// TIA Portal V16 export
// export: Created 2022-03-28T07:44:06.5972207Z, ExportSetting WithDefaults, DisplayName Totally Integrated Automation Portal, DisplayVersion V16 Update 5, DisplayName TIA Portal Version Control Interface, DisplayVersion V16 Update 2, DisplayName TIA Portal Openness, DisplayVersion V16 Update 5, DisplayName STEP 7 Professional, DisplayVersion V16 Update 5, DisplayName STEP 7 Safety, DisplayVersion V16, DisplayName WinCC Professional, DisplayVersion V16 Update 5
FUNCTION_BLOCK "fb_01_Cycle"   // FB1, LAD
{ S7_Optimized_Access := 'TRUE' }
VERSION : 0.1
// stored: AutoNumber false, IsIECCheckEnabled false, IsRetainMemResEnabled false, MemoryReserve 100, SetENOAutomatically false, UDAEnableTagReadback false
   VAR
      TON_Delay : Array[1..10] of TON_TIME;
      TP_Reset { S7_SetPoint := 'True'} : TP_TIME;
   END_VAR
   VAR_TEMP
      bBypassRobot : Bool;
      bRobotReset : Bool;
      bIsInverted : Bool;
   END_VAR
   VAR_TEMP   // added for the SCL form of the ladder/FBD networks
      _w1 : Bool;
      _w2 : Bool;
   END_VAR
BEGIN

REGION Network 1: Reseteo Ciclos por Emergencias
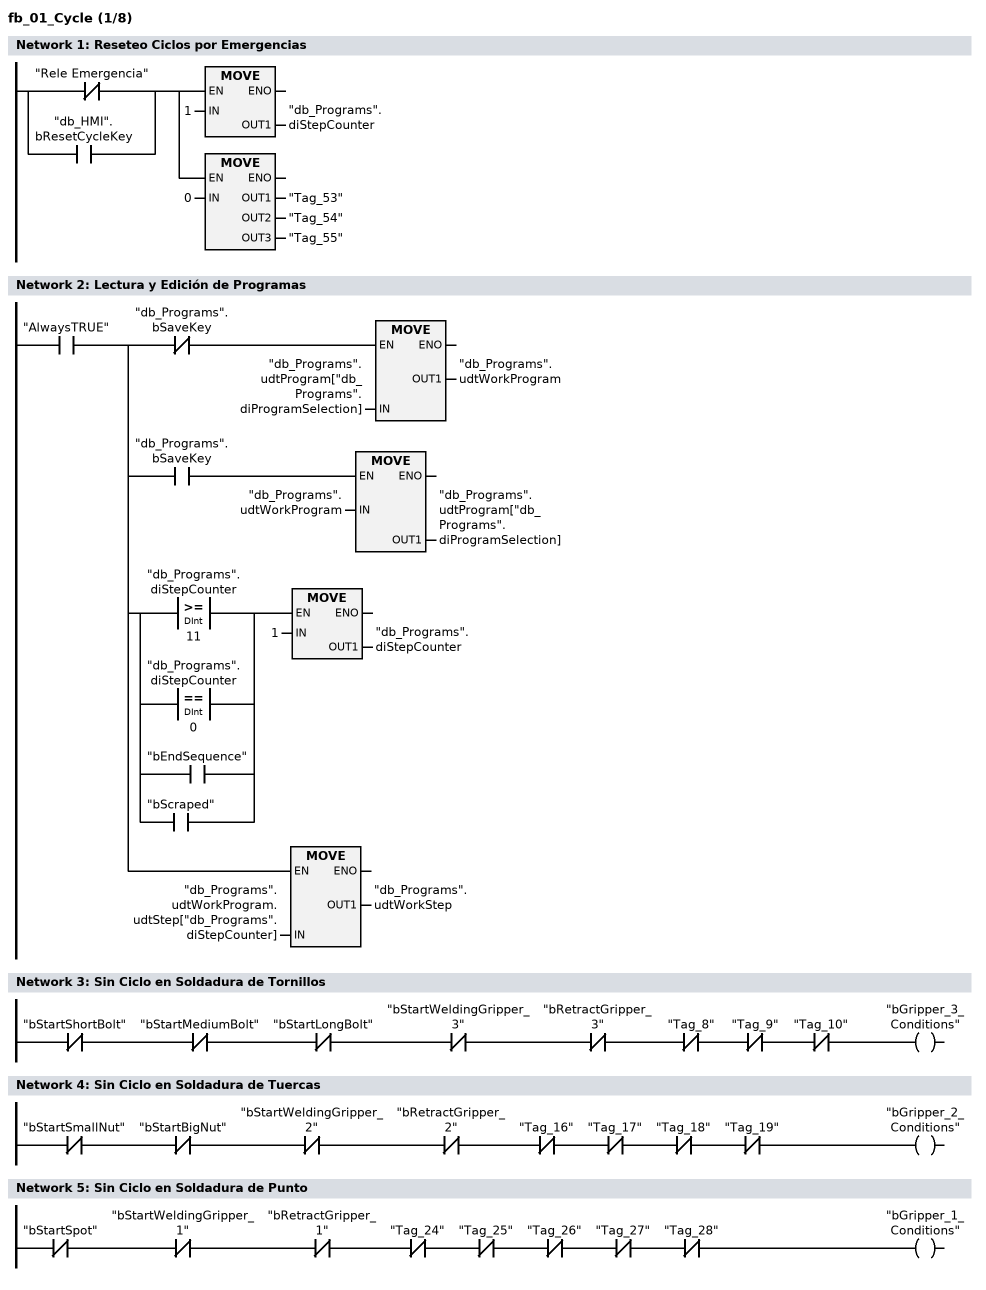
   RUNG wire#powerrail
      I_Contact( "Rele Emergencia" )
      wire#w1
      Move(in := 1, out1 => "db_Programs".diStepCounter)
   END_RUNG
   RUNG wire#powerrail
      Contact( "db_HMI".bResetCycleKey )
   END_RUNG wire#w1
   RUNG wire#w1
      Move(in := 0, out1 => "Tag_53", out2 => "Tag_54", out3 => "Tag_55")
   END_RUNG
   // the same network as SCL:
   IF NOT "Rele Emergencia" OR "db_HMI".bResetCycleKey THEN
       "db_Programs".diStepCounter := 1;
       "Tag_53" := 0;
       "Tag_54" := 0;
       "Tag_55" := 0;
   END_IF;
END_REGION

REGION Network 2: Lectura y Edición de Programas
   RUNG wire#powerrail
      Contact( "AlwaysTRUE" )
      wire#w1
      I_Contact( "db_Programs".bSaveKey )
      Move(in := "db_Programs".udtProgram["db_Programs".diProgramSelection], out1 => "db_Programs".udtWorkProgram)
   END_RUNG
   RUNG wire#w1
      Contact( "db_Programs".bSaveKey )
      Move(in := "db_Programs".udtWorkProgram, out1 => "db_Programs".udtProgram["db_Programs".diProgramSelection])
   END_RUNG
   RUNG wire#w1
      { S7_Templates := "SrcType := DInt" } GE_Contact(in1 := "db_Programs".diStepCounter, in2 := 11)
      wire#w2
      Move(in := 1, out1 => "db_Programs".diStepCounter)
   END_RUNG
   RUNG wire#w1
      { S7_Templates := "SrcType := DInt" } EQ_Contact(in1 := "db_Programs".diStepCounter, in2 := 0)
   END_RUNG wire#w2
   RUNG wire#w1
      Contact( "bEndSequence" )
   END_RUNG wire#w2
   RUNG wire#w1
      Contact( "bScraped" )
   END_RUNG wire#w2
   RUNG wire#w1
      Move(in := "db_Programs".udtWorkProgram.udtStep["db_Programs".diStepCounter], out1 => "db_Programs".udtWorkStep)
   END_RUNG
   // the same network as SCL:
   IF "AlwaysTRUE" AND NOT "db_Programs".bSaveKey THEN
       "db_Programs".udtWorkProgram := "db_Programs".udtProgram["db_Programs".diProgramSelection];
   END_IF;
   IF "AlwaysTRUE" AND "db_Programs".bSaveKey THEN
       "db_Programs".udtProgram["db_Programs".diProgramSelection] := "db_Programs".udtWorkProgram;
   END_IF;
   IF "AlwaysTRUE" AND (("db_Programs".diStepCounter >= 11) OR ("db_Programs".diStepCounter = 0) OR "bEndSequence" OR "bScraped") THEN
       "db_Programs".diStepCounter := 1;
   END_IF;
   IF "AlwaysTRUE" THEN
       "db_Programs".udtWorkStep := "db_Programs".udtWorkProgram.udtStep["db_Programs".diStepCounter];
   END_IF;
END_REGION

REGION Network 3: Sin Ciclo en Soldadura de Tornillos
   RUNG wire#powerrail
      I_Contact( "bStartShortBolt" )
      I_Contact( "bStartMediumBolt" )
      I_Contact( "bStartLongBolt" )
      I_Contact( "bStartWeldingGripper_3" )
      I_Contact( "bRetractGripper_3" )
      I_Contact( "Tag_8" )
      I_Contact( "Tag_9" )
      I_Contact( "Tag_10" )
      Coil( "bGripper_3_Conditions" )
   END_RUNG
   // the same network as SCL:
   "bGripper_3_Conditions" := NOT "bStartShortBolt" AND NOT "bStartMediumBolt" AND NOT "bStartLongBolt" AND NOT "bStartWeldingGripper_3" AND NOT "bRetractGripper_3" AND NOT "Tag_8" AND NOT "Tag_9" AND NOT "Tag_10";
END_REGION

REGION Network 4: Sin Ciclo en Soldadura de Tuercas
   RUNG wire#powerrail
      I_Contact( "bStartSmallNut" )
      I_Contact( "bStartBigNut" )
      I_Contact( "bStartWeldingGripper_2" )
      I_Contact( "bRetractGripper_2" )
      I_Contact( "Tag_16" )
      I_Contact( "Tag_17" )
      I_Contact( "Tag_18" )
      I_Contact( "Tag_19" )
      Coil( "bGripper_2_Conditions" )
   END_RUNG
   // the same network as SCL:
   "bGripper_2_Conditions" := NOT "bStartSmallNut" AND NOT "bStartBigNut" AND NOT "bStartWeldingGripper_2" AND NOT "bRetractGripper_2" AND NOT "Tag_16" AND NOT "Tag_17" AND NOT "Tag_18" AND NOT "Tag_19";
END_REGION

REGION Network 5: Sin Ciclo en Soldadura de Punto
   RUNG wire#powerrail
      I_Contact( "bStartSpot" )
      I_Contact( "bStartWeldingGripper_1" )
      I_Contact( "bRetractGripper_1" )
      I_Contact( "Tag_24" )
      I_Contact( "Tag_25" )
      I_Contact( "Tag_26" )
      I_Contact( "Tag_27" )
      I_Contact( "Tag_28" )
      Coil( "bGripper_1_Conditions" )
   END_RUNG
   // the same network as SCL:
   "bGripper_1_Conditions" := NOT "bStartSpot" AND NOT "bStartWeldingGripper_1" AND NOT "bRetractGripper_1" AND NOT "Tag_24" AND NOT "Tag_25" AND NOT "Tag_26" AND NOT "Tag_27" AND NOT "Tag_28";
END_REGION

REGION Network 6: Condiciones Ciclo Auxiliares
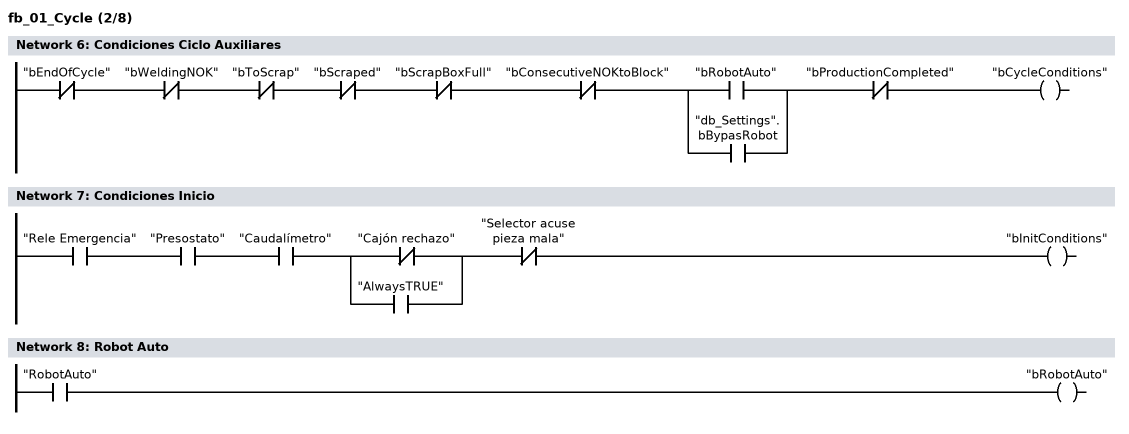
   RUNG wire#powerrail
      I_Contact( "bEndOfCycle" )
      I_Contact( "bWeldingNOK" )
      I_Contact( "bToScrap" )
      I_Contact( "bScraped" )
      I_Contact( "bScrapBoxFull" )
      I_Contact( "bConsecutiveNOKtoBlock" )
      wire#w1
      Contact( "bRobotAuto" )
      wire#w2
      I_Contact( "bProductionCompleted" )
      Coil( "bCycleConditions" )
   END_RUNG
   RUNG wire#w1
      Contact( "db_Settings".bBypasRobot )
   END_RUNG wire#w2
   // the same network as SCL:
   "bCycleConditions" := NOT "bEndOfCycle" AND NOT "bWeldingNOK" AND NOT "bToScrap" AND NOT "bScraped" AND NOT "bScrapBoxFull" AND NOT "bConsecutiveNOKtoBlock" AND ("bRobotAuto" OR "db_Settings".bBypasRobot) AND NOT "bProductionCompleted";
END_REGION

REGION Network 7: Condiciones Inicio
   RUNG wire#powerrail
      Contact( "Rele Emergencia" )
      Contact( "Presostato" )
      Contact( "Caudalímetro" )
      wire#w1
      I_Contact( "Cajón rechazo" )
      wire#w2
      I_Contact( "Selector acuse pieza mala" )
      Coil( "bInitConditions" )
   END_RUNG
   RUNG wire#w1
      Contact( "AlwaysTRUE" )
   END_RUNG wire#w2
   // the same network as SCL:
   "bInitConditions" := "Rele Emergencia" AND "Presostato" AND "Caudalímetro" AND (NOT "Cajón rechazo" OR "AlwaysTRUE") AND NOT "Selector acuse pieza mala";
END_REGION

REGION Network 8: Robot Auto
   RUNG wire#powerrail
      Contact( "RobotAuto" )
      Coil( "bRobotAuto" )
   END_RUNG
   // the same network as SCL:
   "bRobotAuto" := "RobotAuto";
END_REGION

REGION Network 9: Selección Acción
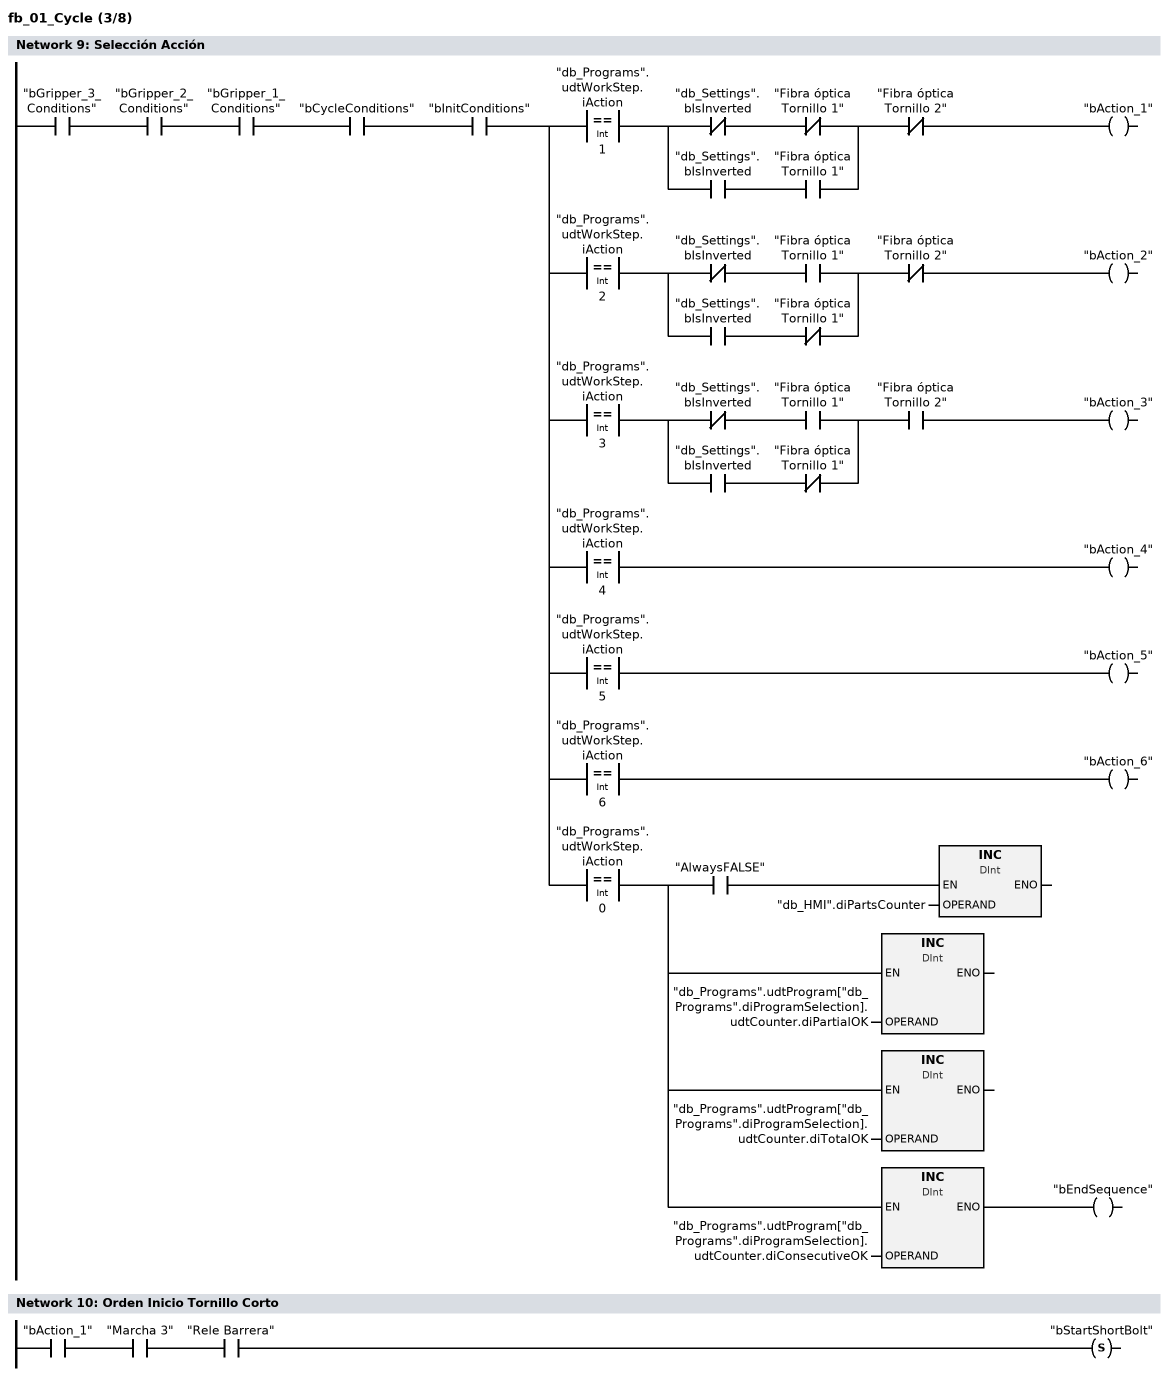
   RUNG wire#powerrail
      Contact( "bGripper_3_Conditions" )
      Contact( "bGripper_2_Conditions" )
      Contact( "bGripper_1_Conditions" )
      Contact( "bCycleConditions" )
      Contact( "bInitConditions" )
      wire#w1
      { S7_Templates := "SrcType := Int" } EQ_Contact(in1 := "db_Programs".udtWorkStep.iAction, in2 := 1)
      wire#w2
      I_Contact( "db_Settings".bIsInverted )
      I_Contact( "Fibra óptica Tornillo 1" )
      wire#w3
      I_Contact( "Fibra óptica Tornillo 2" )
      Coil( "bAction_1" )
   END_RUNG
   RUNG wire#w2
      Contact( "db_Settings".bIsInverted )
      Contact( "Fibra óptica Tornillo 1" )
   END_RUNG wire#w3
   RUNG wire#w1
      { S7_Templates := "SrcType := Int" } EQ_Contact(in1 := "db_Programs".udtWorkStep.iAction, in2 := 2)
      wire#w4
      I_Contact( "db_Settings".bIsInverted )
      Contact( "Fibra óptica Tornillo 1" )
      wire#w5
      I_Contact( "Fibra óptica Tornillo 2" )
      Coil( "bAction_2" )
   END_RUNG
   RUNG wire#w4
      Contact( "db_Settings".bIsInverted )
      I_Contact( "Fibra óptica Tornillo 1" )
   END_RUNG wire#w5
   RUNG wire#w1
      { S7_Templates := "SrcType := Int" } EQ_Contact(in1 := "db_Programs".udtWorkStep.iAction, in2 := 3)
      wire#w6
      I_Contact( "db_Settings".bIsInverted )
      Contact( "Fibra óptica Tornillo 1" )
      wire#w7
      Contact( "Fibra óptica Tornillo 2" )
      Coil( "bAction_3" )
   END_RUNG
   RUNG wire#w6
      Contact( "db_Settings".bIsInverted )
      I_Contact( "Fibra óptica Tornillo 1" )
   END_RUNG wire#w7
   RUNG wire#w1
      { S7_Templates := "SrcType := Int" } EQ_Contact(in1 := "db_Programs".udtWorkStep.iAction, in2 := 4)
      Coil( "bAction_4" )
   END_RUNG
   RUNG wire#w1
      { S7_Templates := "SrcType := Int" } EQ_Contact(in1 := "db_Programs".udtWorkStep.iAction, in2 := 5)
      Coil( "bAction_5" )
   END_RUNG
   RUNG wire#w1
      { S7_Templates := "SrcType := Int" } EQ_Contact(in1 := "db_Programs".udtWorkStep.iAction, in2 := 6)
      Coil( "bAction_6" )
   END_RUNG
   RUNG wire#w1
      { S7_Templates := "SrcType := Int" } EQ_Contact(in1 := "db_Programs".udtWorkStep.iAction, in2 := 0)
      wire#w8
      Contact( "AlwaysFALSE" )
      { S7_Templates := "DestType := DInt" } Inc( "db_HMI".diPartsCounter )
   END_RUNG
   RUNG wire#w8
      { S7_Templates := "DestType := DInt" } Inc( "db_Programs".udtProgram["db_Programs".diProgramSelection].udtCounter.diPartialOK )
   END_RUNG
   RUNG wire#w8
      { S7_Templates := "DestType := DInt" } Inc( "db_Programs".udtProgram["db_Programs".diProgramSelection].udtCounter.diTotalOK )
   END_RUNG
   RUNG wire#w8
      { S7_Templates := "DestType := DInt" } Inc( "db_Programs".udtProgram["db_Programs".diProgramSelection].udtCounter.diConsecutiveOK )
      Coil( "bEndSequence" )
   END_RUNG
   // the same network as SCL:
   #_w1 := "bGripper_3_Conditions" AND "bGripper_2_Conditions" AND "bGripper_1_Conditions" AND "bCycleConditions" AND "bInitConditions";
   "bAction_1" := #_w1 AND ("db_Programs".udtWorkStep.iAction = 1) AND ((NOT "db_Settings".bIsInverted AND NOT "Fibra óptica Tornillo 1") OR ("db_Settings".bIsInverted AND "Fibra óptica Tornillo 1")) AND NOT "Fibra óptica Tornillo 2";
   "bAction_2" := #_w1 AND ("db_Programs".udtWorkStep.iAction = 2) AND ((NOT "db_Settings".bIsInverted AND "Fibra óptica Tornillo 1") OR ("db_Settings".bIsInverted AND NOT "Fibra óptica Tornillo 1")) AND NOT "Fibra óptica Tornillo 2";
   "bAction_3" := #_w1 AND ("db_Programs".udtWorkStep.iAction = 3) AND ((NOT "db_Settings".bIsInverted AND "Fibra óptica Tornillo 1") OR ("db_Settings".bIsInverted AND NOT "Fibra óptica Tornillo 1")) AND "Fibra óptica Tornillo 2";
   "bAction_4" := #_w1 AND ("db_Programs".udtWorkStep.iAction = 4);
   "bAction_5" := #_w1 AND ("db_Programs".udtWorkStep.iAction = 5);
   "bAction_6" := #_w1 AND ("db_Programs".udtWorkStep.iAction = 6);
   #_w2 := #_w1 AND ("db_Programs".udtWorkStep.iAction = 0);
   IF #_w2 AND "AlwaysFALSE" THEN "db_HMI".diPartsCounter := "db_HMI".diPartsCounter + 1; END_IF;
   IF #_w2 THEN
       "db_Programs".udtProgram["db_Programs".diProgramSelection].udtCounter.diPartialOK := "db_Programs".udtProgram["db_Programs".diProgramSelection].udtCounter.diPartialOK + 1;
       "db_Programs".udtProgram["db_Programs".diProgramSelection].udtCounter.diTotalOK := "db_Programs".udtProgram["db_Programs".diProgramSelection].udtCounter.diTotalOK + 1;
       "db_Programs".udtProgram["db_Programs".diProgramSelection].udtCounter.diConsecutiveOK := "db_Programs".udtProgram["db_Programs".diProgramSelection].udtCounter.diConsecutiveOK + 1;
   END_IF;
   "bEndSequence" := #_w2;
END_REGION

REGION Network 10: Orden Inicio Tornillo Corto
   RUNG wire#powerrail
      Contact( "bAction_1" )
      Contact( "Marcha 3" )
      Contact( "Rele Barrera" )
      S_Coil( "bStartShortBolt" )
   END_RUNG
   // the same network as SCL:
   IF "bAction_1" AND "Marcha 3" AND "Rele Barrera" THEN "bStartShortBolt" := TRUE; END_IF;
END_REGION

REGION Network 11: Orden Inicio Tornillo Mediano
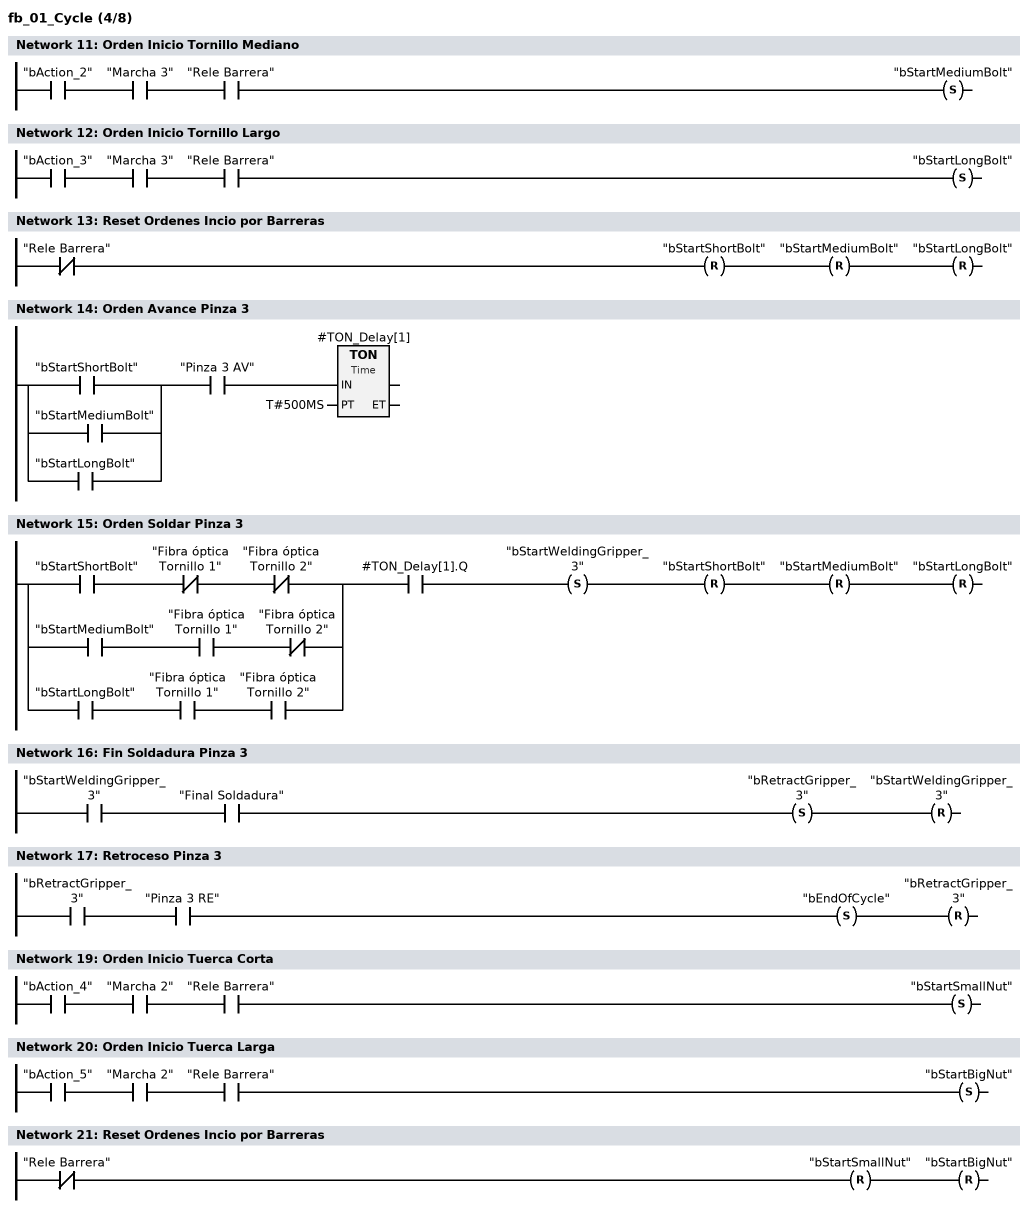
   RUNG wire#powerrail
      Contact( "bAction_2" )
      Contact( "Marcha 3" )
      Contact( "Rele Barrera" )
      S_Coil( "bStartMediumBolt" )
   END_RUNG
   // the same network as SCL:
   IF "bAction_2" AND "Marcha 3" AND "Rele Barrera" THEN "bStartMediumBolt" := TRUE; END_IF;
END_REGION

REGION Network 12: Orden Inicio Tornillo Largo
   RUNG wire#powerrail
      Contact( "bAction_3" )
      Contact( "Marcha 3" )
      Contact( "Rele Barrera" )
      S_Coil( "bStartLongBolt" )
   END_RUNG
   // the same network as SCL:
   IF "bAction_3" AND "Marcha 3" AND "Rele Barrera" THEN "bStartLongBolt" := TRUE; END_IF;
END_REGION

REGION Network 13: Reset Ordenes Incio por Barreras
   RUNG wire#powerrail
      I_Contact( "Rele Barrera" )
      R_Coil( "bStartShortBolt" )
      R_Coil( "bStartMediumBolt" )
      R_Coil( "bStartLongBolt" )
   END_RUNG
   // the same network as SCL:
   IF NOT "Rele Barrera" THEN
       "bStartShortBolt" := FALSE;
       "bStartMediumBolt" := FALSE;
       "bStartLongBolt" := FALSE;
   END_IF;
END_REGION

REGION Network 14: Orden Avance Pinza 3
   RUNG wire#powerrail
      Contact( "bStartShortBolt" )
      wire#w1
      Contact( "Pinza 3 AV" )
      { S7_Templates := "time_type := Time" } #TON_Delay[1].TON(pt := T#500MS, et =>)
   END_RUNG
   RUNG wire#powerrail
      Contact( "bStartMediumBolt" )
   END_RUNG wire#w1
   RUNG wire#powerrail
      Contact( "bStartLongBolt" )
   END_RUNG wire#w1
   // the same network as SCL:
   #TON_Delay[1].TON(IN := ("bStartShortBolt" OR "bStartMediumBolt" OR "bStartLongBolt") AND "Pinza 3 AV",
                     PT := T#500MS);
END_REGION

REGION Network 15: Orden Soldar Pinza 3
   RUNG wire#powerrail
      Contact( "bStartShortBolt" )
      I_Contact( "Fibra óptica Tornillo 1" )
      I_Contact( "Fibra óptica Tornillo 2" )
      wire#w1
      Contact( #TON_Delay[1].Q )
      S_Coil( "bStartWeldingGripper_3" )
      R_Coil( "bStartShortBolt" )
      R_Coil( "bStartMediumBolt" )
      R_Coil( "bStartLongBolt" )
   END_RUNG
   RUNG wire#powerrail
      Contact( "bStartMediumBolt" )
      Contact( "Fibra óptica Tornillo 1" )
      I_Contact( "Fibra óptica Tornillo 2" )
   END_RUNG wire#w1
   RUNG wire#powerrail
      Contact( "bStartLongBolt" )
      Contact( "Fibra óptica Tornillo 1" )
      Contact( "Fibra óptica Tornillo 2" )
   END_RUNG wire#w1
   // the same network as SCL:
   IF (("bStartShortBolt" AND NOT "Fibra óptica Tornillo 1" AND NOT "Fibra óptica Tornillo 2") OR ("bStartMediumBolt" AND "Fibra óptica Tornillo 1" AND NOT "Fibra óptica Tornillo 2") OR ("bStartLongBolt" AND "Fibra óptica Tornillo 1" AND "Fibra óptica Tornillo 2")) AND #TON_Delay[1].Q THEN
       "bStartWeldingGripper_3" := TRUE;
   END_IF;
   #_w1 := (("bStartShortBolt" AND NOT "Fibra óptica Tornillo 1" AND NOT "Fibra óptica Tornillo 2") OR ("bStartMediumBolt" AND "Fibra óptica Tornillo 1" AND NOT "Fibra óptica Tornillo 2") OR ("bStartLongBolt" AND "Fibra óptica Tornillo 1" AND "Fibra óptica Tornillo 2")) AND #TON_Delay[1].Q;
   IF #_w1 THEN
       "bStartShortBolt" := FALSE;
       "bStartMediumBolt" := FALSE;
       "bStartLongBolt" := FALSE;
   END_IF;
END_REGION

REGION Network 16: Fin Soldadura Pinza 3
   RUNG wire#powerrail
      Contact( "bStartWeldingGripper_3" )
      Contact( "Final Soldadura" )
      S_Coil( "bRetractGripper_3" )
      R_Coil( "bStartWeldingGripper_3" )
   END_RUNG
   // the same network as SCL:
   IF "bStartWeldingGripper_3" AND "Final Soldadura" THEN
       "bRetractGripper_3" := TRUE;
       "bStartWeldingGripper_3" := FALSE;
   END_IF;
END_REGION

REGION Network 17: Retroceso Pinza 3
   RUNG wire#powerrail
      Contact( "bRetractGripper_3" )
      Contact( "Pinza 3 RE" )
      S_Coil( "bEndOfCycle" )
      R_Coil( "bRetractGripper_3" )
   END_RUNG
   // the same network as SCL:
   IF "bRetractGripper_3" AND "Pinza 3 RE" THEN
       "bEndOfCycle" := TRUE;
       "bRetractGripper_3" := FALSE;
   END_IF;
END_REGION

REGION Network 19: Orden Inicio Tuerca Corta
   RUNG wire#powerrail
      Contact( "bAction_4" )
      Contact( "Marcha 2" )
      Contact( "Rele Barrera" )
      S_Coil( "bStartSmallNut" )
   END_RUNG
   // the same network as SCL:
   IF "bAction_4" AND "Marcha 2" AND "Rele Barrera" THEN "bStartSmallNut" := TRUE; END_IF;
END_REGION

REGION Network 20: Orden Inicio Tuerca Larga
   RUNG wire#powerrail
      Contact( "bAction_5" )
      Contact( "Marcha 2" )
      Contact( "Rele Barrera" )
      S_Coil( "bStartBigNut" )
   END_RUNG
   // the same network as SCL:
   IF "bAction_5" AND "Marcha 2" AND "Rele Barrera" THEN "bStartBigNut" := TRUE; END_IF;
END_REGION

REGION Network 21: Reset Ordenes Incio por Barreras
   RUNG wire#powerrail
      I_Contact( "Rele Barrera" )
      R_Coil( "bStartSmallNut" )
      R_Coil( "bStartBigNut" )
   END_RUNG
   // the same network as SCL:
   IF NOT "Rele Barrera" THEN
       "bStartSmallNut" := FALSE;
       "bStartBigNut" := FALSE;
   END_IF;
END_REGION

REGION Network 22: Orden Bajar y Soldar Pinza 2
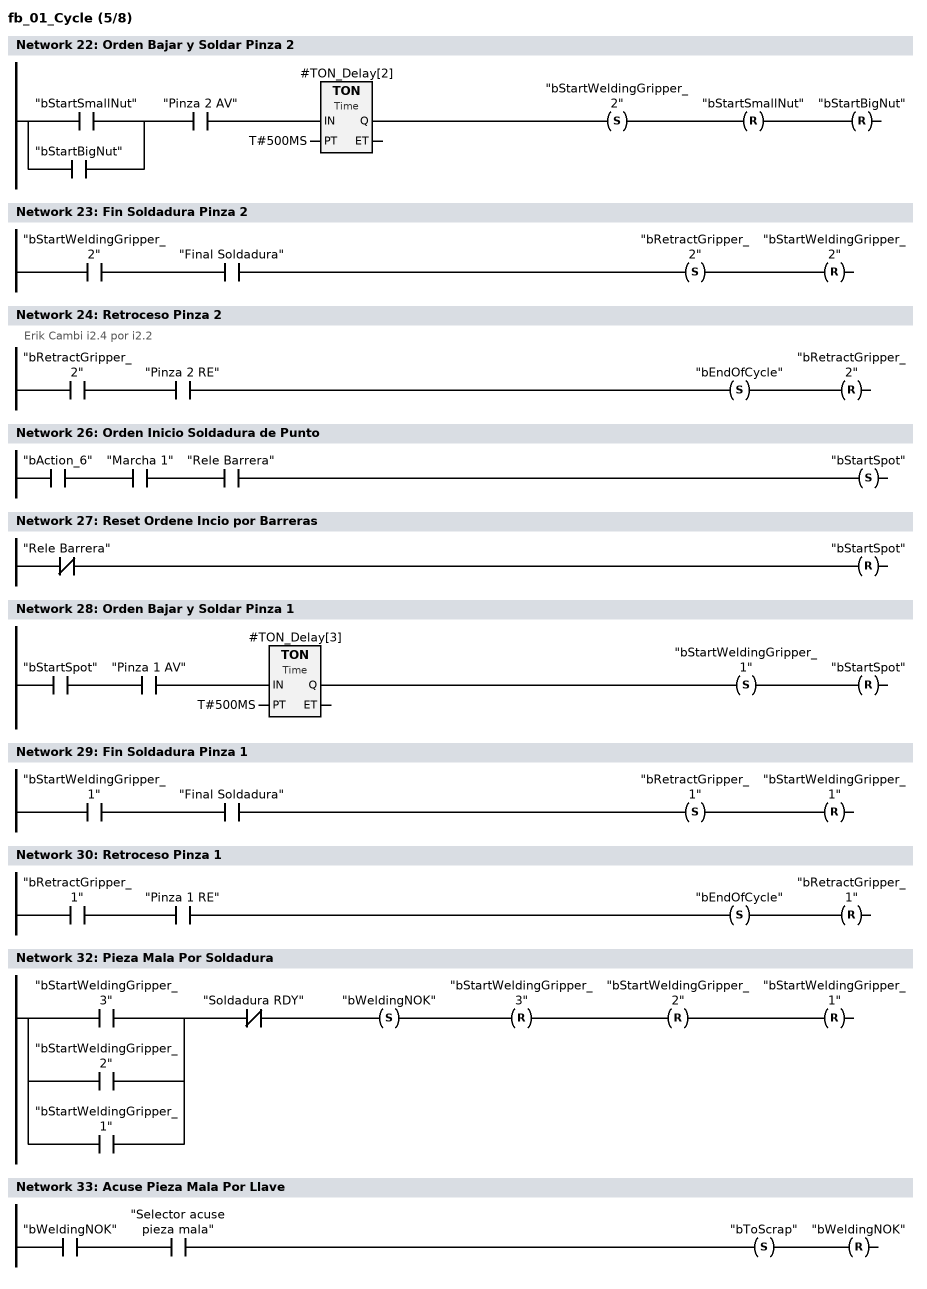
   RUNG wire#powerrail
      Contact( "bStartSmallNut" )
      wire#w1
      Contact( "Pinza 2 AV" )
      { S7_Templates := "time_type := Time" } #TON_Delay[2].TON(pt := T#500MS, et =>)
      S_Coil( "bStartWeldingGripper_2" )
      R_Coil( "bStartSmallNut" )
      R_Coil( "bStartBigNut" )
   END_RUNG
   RUNG wire#powerrail
      Contact( "bStartBigNut" )
   END_RUNG wire#w1
   // the same network as SCL:
   #TON_Delay[2].TON(IN := ("bStartSmallNut" OR "bStartBigNut") AND "Pinza 2 AV", PT := T#500MS);
   IF #TON_Delay[2].Q THEN
       "bStartWeldingGripper_2" := TRUE;
       "bStartSmallNut" := FALSE;
       "bStartBigNut" := FALSE;
   END_IF;
END_REGION

REGION Network 23: Fin Soldadura Pinza 2
   RUNG wire#powerrail
      Contact( "bStartWeldingGripper_2" )
      Contact( "Final Soldadura" )
      S_Coil( "bRetractGripper_2" )
      R_Coil( "bStartWeldingGripper_2" )
   END_RUNG
   // the same network as SCL:
   IF "bStartWeldingGripper_2" AND "Final Soldadura" THEN
       "bRetractGripper_2" := TRUE;
       "bStartWeldingGripper_2" := FALSE;
   END_IF;
END_REGION

REGION Network 24: Retroceso Pinza 2
   // Erik Cambi i2.4 por i2.2
   RUNG wire#powerrail
      Contact( "bRetractGripper_2" )
      Contact( "Pinza 2 RE" )
      S_Coil( "bEndOfCycle" )
      R_Coil( "bRetractGripper_2" )
   END_RUNG
   // the same network as SCL:
   IF "bRetractGripper_2" AND "Pinza 2 RE" THEN
       "bEndOfCycle" := TRUE;
       "bRetractGripper_2" := FALSE;
   END_IF;
END_REGION

REGION Network 26: Orden Inicio Soldadura de Punto
   RUNG wire#powerrail
      Contact( "bAction_6" )
      Contact( "Marcha 1" )
      Contact( "Rele Barrera" )
      S_Coil( "bStartSpot" )
   END_RUNG
   // the same network as SCL:
   IF "bAction_6" AND "Marcha 1" AND "Rele Barrera" THEN "bStartSpot" := TRUE; END_IF;
END_REGION

REGION Network 27: Reset Ordene Incio por Barreras
   RUNG wire#powerrail
      I_Contact( "Rele Barrera" )
      R_Coil( "bStartSpot" )
   END_RUNG
   // the same network as SCL:
   IF NOT "Rele Barrera" THEN "bStartSpot" := FALSE; END_IF;
END_REGION

REGION Network 28: Orden Bajar y Soldar Pinza 1
   RUNG wire#powerrail
      Contact( "bStartSpot" )
      Contact( "Pinza 1 AV" )
      { S7_Templates := "time_type := Time" } #TON_Delay[3].TON(pt := T#500MS, et =>)
      S_Coil( "bStartWeldingGripper_1" )
      R_Coil( "bStartSpot" )
   END_RUNG
   // the same network as SCL:
   #TON_Delay[3].TON(IN := "bStartSpot" AND "Pinza 1 AV", PT := T#500MS);
   IF #TON_Delay[3].Q THEN
       "bStartWeldingGripper_1" := TRUE;
       "bStartSpot" := FALSE;
   END_IF;
END_REGION

REGION Network 29: Fin Soldadura Pinza 1
   RUNG wire#powerrail
      Contact( "bStartWeldingGripper_1" )
      Contact( "Final Soldadura" )
      S_Coil( "bRetractGripper_1" )
      R_Coil( "bStartWeldingGripper_1" )
   END_RUNG
   // the same network as SCL:
   IF "bStartWeldingGripper_1" AND "Final Soldadura" THEN
       "bRetractGripper_1" := TRUE;
       "bStartWeldingGripper_1" := FALSE;
   END_IF;
END_REGION

REGION Network 30: Retroceso Pinza 1
   RUNG wire#powerrail
      Contact( "bRetractGripper_1" )
      Contact( "Pinza 1 RE" )
      S_Coil( "bEndOfCycle" )
      R_Coil( "bRetractGripper_1" )
   END_RUNG
   // the same network as SCL:
   IF "bRetractGripper_1" AND "Pinza 1 RE" THEN
       "bEndOfCycle" := TRUE;
       "bRetractGripper_1" := FALSE;
   END_IF;
END_REGION

REGION Network 32: Pieza Mala Por Soldadura
   RUNG wire#powerrail
      Contact( "bStartWeldingGripper_3" )
      wire#w1
      I_Contact( "Soldadura RDY" )
      S_Coil( "bWeldingNOK" )
      R_Coil( "bStartWeldingGripper_3" )
      R_Coil( "bStartWeldingGripper_2" )
      R_Coil( "bStartWeldingGripper_1" )
   END_RUNG
   RUNG wire#powerrail
      Contact( "bStartWeldingGripper_2" )
   END_RUNG wire#w1
   RUNG wire#powerrail
      Contact( "bStartWeldingGripper_1" )
   END_RUNG wire#w1
   // the same network as SCL:
   IF ("bStartWeldingGripper_3" OR "bStartWeldingGripper_2" OR "bStartWeldingGripper_1") AND NOT "Soldadura RDY" THEN
       "bWeldingNOK" := TRUE;
   END_IF;
   #_w1 := ("bStartWeldingGripper_3" OR "bStartWeldingGripper_2" OR "bStartWeldingGripper_1") AND NOT "Soldadura RDY";
   IF #_w1 THEN
       "bStartWeldingGripper_3" := FALSE;
       "bStartWeldingGripper_2" := FALSE;
       "bStartWeldingGripper_1" := FALSE;
   END_IF;
END_REGION

REGION Network 33: Acuse Pieza Mala Por Llave
   RUNG wire#powerrail
      Contact( "bWeldingNOK" )
      Contact( "Selector acuse pieza mala" )
      S_Coil( "bToScrap" )
      R_Coil( "bWeldingNOK" )
   END_RUNG
   // the same network as SCL:
   IF "bWeldingNOK" AND "Selector acuse pieza mala" THEN
       "bToScrap" := TRUE;
       "bWeldingNOK" := FALSE;
   END_IF;
END_REGION

REGION Network 34: Desechar Pieza Mala
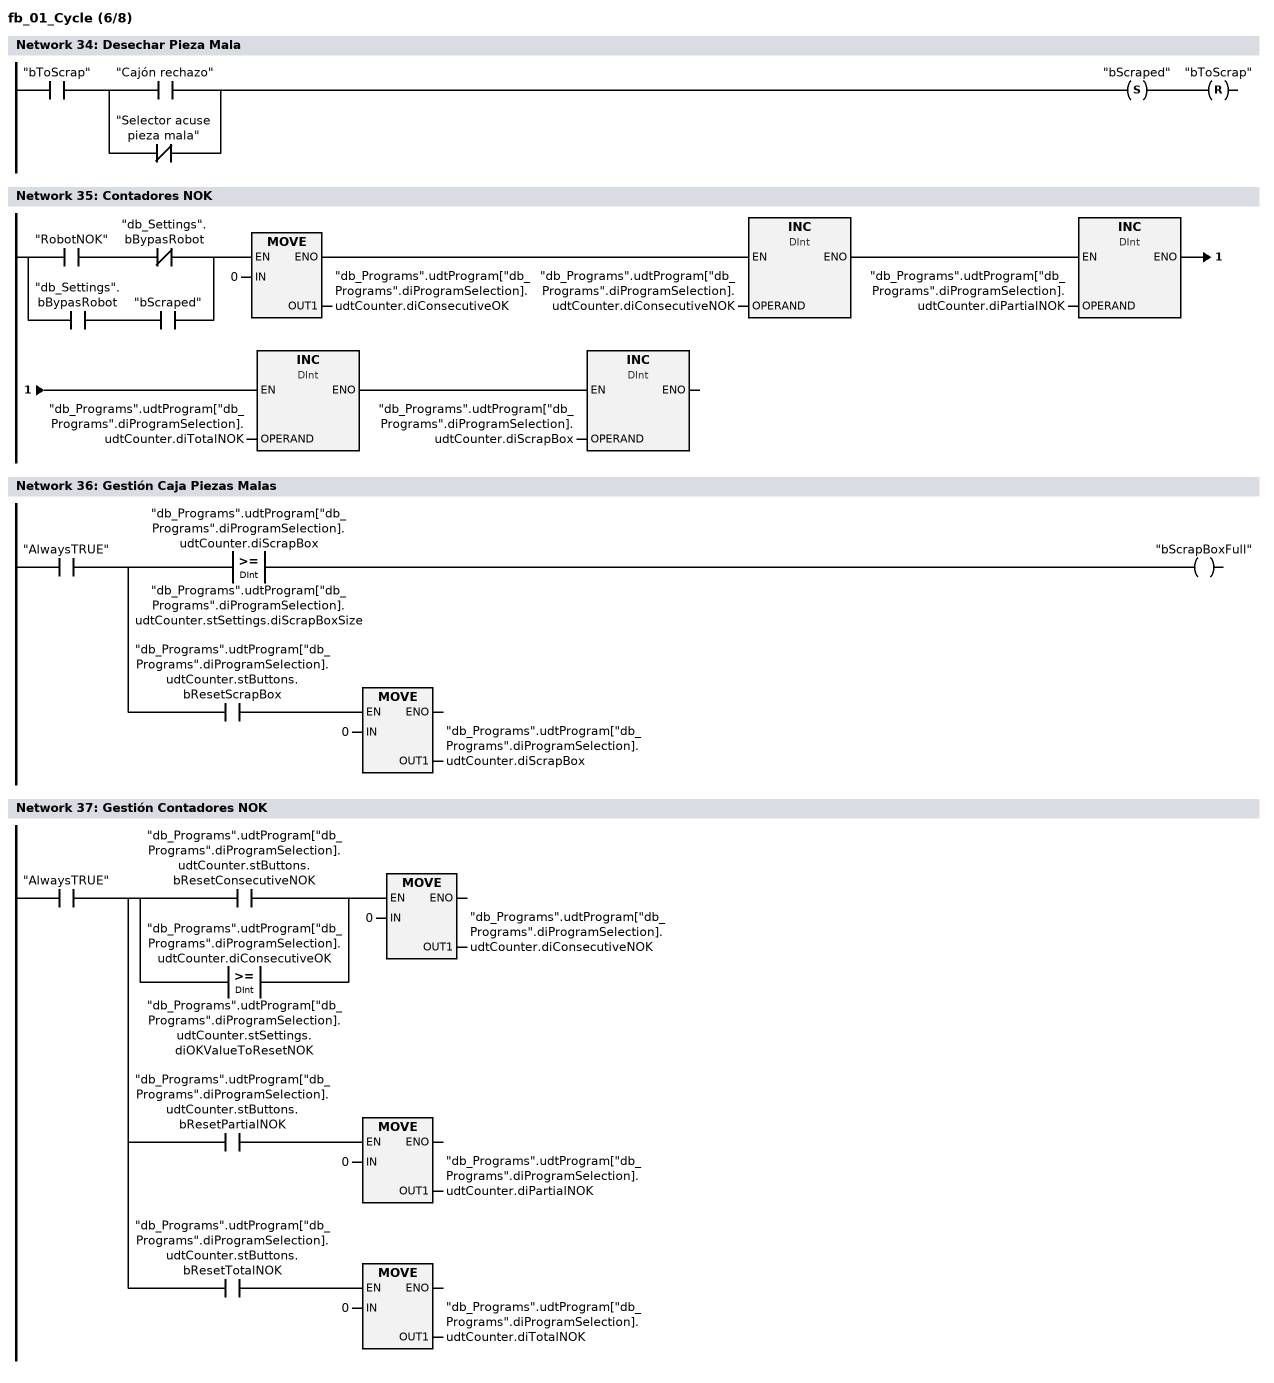
   RUNG wire#powerrail
      Contact( "bToScrap" )
      wire#w1
      Contact( "Cajón rechazo" )
      wire#w2
      S_Coil( "bScraped" )
      R_Coil( "bToScrap" )
   END_RUNG
   RUNG wire#w1
      I_Contact( "Selector acuse pieza mala" )
   END_RUNG wire#w2
   // the same network as SCL:
   IF "bToScrap" AND ("Cajón rechazo" OR NOT "Selector acuse pieza mala") THEN
       "bScraped" := TRUE;
       "bToScrap" := FALSE;
   END_IF;
END_REGION

REGION Network 35: Contadores NOK
   RUNG wire#powerrail
      Contact( "RobotNOK" )
      I_Contact( "db_Settings".bBypasRobot )
      wire#w1
      Move(in := 0, out1 => "db_Programs".udtProgram["db_Programs".diProgramSelection].udtCounter.diConsecutiveOK)
      { S7_Templates := "DestType := DInt" } Inc( "db_Programs".udtProgram["db_Programs".diProgramSelection].udtCounter.diConsecutiveNOK )
      { S7_Templates := "DestType := DInt" } Inc( "db_Programs".udtProgram["db_Programs".diProgramSelection].udtCounter.diPartialNOK )
      { S7_Templates := "DestType := DInt" } Inc( "db_Programs".udtProgram["db_Programs".diProgramSelection].udtCounter.diTotalNOK )
      { S7_Templates := "DestType := DInt" } Inc( "db_Programs".udtProgram["db_Programs".diProgramSelection].udtCounter.diScrapBox )
   END_RUNG
   RUNG wire#powerrail
      Contact( "db_Settings".bBypasRobot )
      Contact( "bScraped" )
   END_RUNG wire#w1
   // the same network as SCL:
   IF ("RobotNOK" AND NOT "db_Settings".bBypasRobot) OR ("db_Settings".bBypasRobot AND "bScraped") THEN
       "db_Programs".udtProgram["db_Programs".diProgramSelection].udtCounter.diConsecutiveOK := 0;
       "db_Programs".udtProgram["db_Programs".diProgramSelection].udtCounter.diConsecutiveNOK := "db_Programs".udtProgram["db_Programs".diProgramSelection].udtCounter.diConsecutiveNOK + 1;
       "db_Programs".udtProgram["db_Programs".diProgramSelection].udtCounter.diPartialNOK := "db_Programs".udtProgram["db_Programs".diProgramSelection].udtCounter.diPartialNOK + 1;
       "db_Programs".udtProgram["db_Programs".diProgramSelection].udtCounter.diTotalNOK := "db_Programs".udtProgram["db_Programs".diProgramSelection].udtCounter.diTotalNOK + 1;
       "db_Programs".udtProgram["db_Programs".diProgramSelection].udtCounter.diScrapBox := "db_Programs".udtProgram["db_Programs".diProgramSelection].udtCounter.diScrapBox + 1;
   END_IF;
END_REGION

REGION Network 36: Gestión Caja Piezas Malas
   RUNG wire#powerrail
      Contact( "AlwaysTRUE" )
      wire#w1
      { S7_Templates := "SrcType := DInt" } GE_Contact(in1 := "db_Programs".udtProgram["db_Programs".diProgramSelection].udtCounter.diScrapBox, in2 := "db_Programs".udtProgram["db_Programs".diProgramSelection].udtCounter.stSettings.diScrapBoxSize)
      Coil( "bScrapBoxFull" )
   END_RUNG
   RUNG wire#w1
      Contact( "db_Programs".udtProgram["db_Programs".diProgramSelection].udtCounter.stButtons.bResetScrapBox )
      Move(in := 0, out1 => "db_Programs".udtProgram["db_Programs".diProgramSelection].udtCounter.diScrapBox)
   END_RUNG
   // the same network as SCL:
   "bScrapBoxFull" := "AlwaysTRUE" AND ("db_Programs".udtProgram["db_Programs".diProgramSelection].udtCounter.diScrapBox >= "db_Programs".udtProgram["db_Programs".diProgramSelection].udtCounter.stSettings.diScrapBoxSize);
   IF "AlwaysTRUE" AND "db_Programs".udtProgram["db_Programs".diProgramSelection].udtCounter.stButtons.bResetScrapBox THEN
       "db_Programs".udtProgram["db_Programs".diProgramSelection].udtCounter.diScrapBox := 0;
   END_IF;
END_REGION

REGION Network 37: Gestión Contadores NOK
   RUNG wire#powerrail
      Contact( "AlwaysTRUE" )
      wire#w1
      Contact( "db_Programs".udtProgram["db_Programs".diProgramSelection].udtCounter.stButtons.bResetConsecutiveNOK )
      wire#w2
      Move(in := 0, out1 => "db_Programs".udtProgram["db_Programs".diProgramSelection].udtCounter.diConsecutiveNOK)
   END_RUNG
   RUNG wire#w1
      { S7_Templates := "SrcType := DInt" } GE_Contact(in1 := "db_Programs".udtProgram["db_Programs".diProgramSelection].udtCounter.diConsecutiveOK, in2 := "db_Programs".udtProgram["db_Programs".diProgramSelection].udtCounter.stSettings.diOKValueToResetNOK)
   END_RUNG wire#w2
   RUNG wire#w1
      Contact( "db_Programs".udtProgram["db_Programs".diProgramSelection].udtCounter.stButtons.bResetPartialNOK )
      Move(in := 0, out1 => "db_Programs".udtProgram["db_Programs".diProgramSelection].udtCounter.diPartialNOK)
   END_RUNG
   RUNG wire#w1
      Contact( "db_Programs".udtProgram["db_Programs".diProgramSelection].udtCounter.stButtons.bResetTotalNOK )
      Move(in := 0, out1 => "db_Programs".udtProgram["db_Programs".diProgramSelection].udtCounter.diTotalNOK)
   END_RUNG
   // the same network as SCL:
   IF "AlwaysTRUE" AND ("db_Programs".udtProgram["db_Programs".diProgramSelection].udtCounter.stButtons.bResetConsecutiveNOK OR ("db_Programs".udtProgram["db_Programs".diProgramSelection].udtCounter.diConsecutiveOK >= "db_Programs".udtProgram["db_Programs".diProgramSelection].udtCounter.stSettings.diOKValueToResetNOK)) THEN
       "db_Programs".udtProgram["db_Programs".diProgramSelection].udtCounter.diConsecutiveNOK := 0;
   END_IF;
   IF "AlwaysTRUE" AND "db_Programs".udtProgram["db_Programs".diProgramSelection].udtCounter.stButtons.bResetPartialNOK THEN
       "db_Programs".udtProgram["db_Programs".diProgramSelection].udtCounter.diPartialNOK := 0;
   END_IF;
   IF "AlwaysTRUE" AND "db_Programs".udtProgram["db_Programs".diProgramSelection].udtCounter.stButtons.bResetTotalNOK THEN
       "db_Programs".udtProgram["db_Programs".diProgramSelection].udtCounter.diTotalNOK := 0;
   END_IF;
END_REGION

REGION Network 38: Contadores Piezas OK
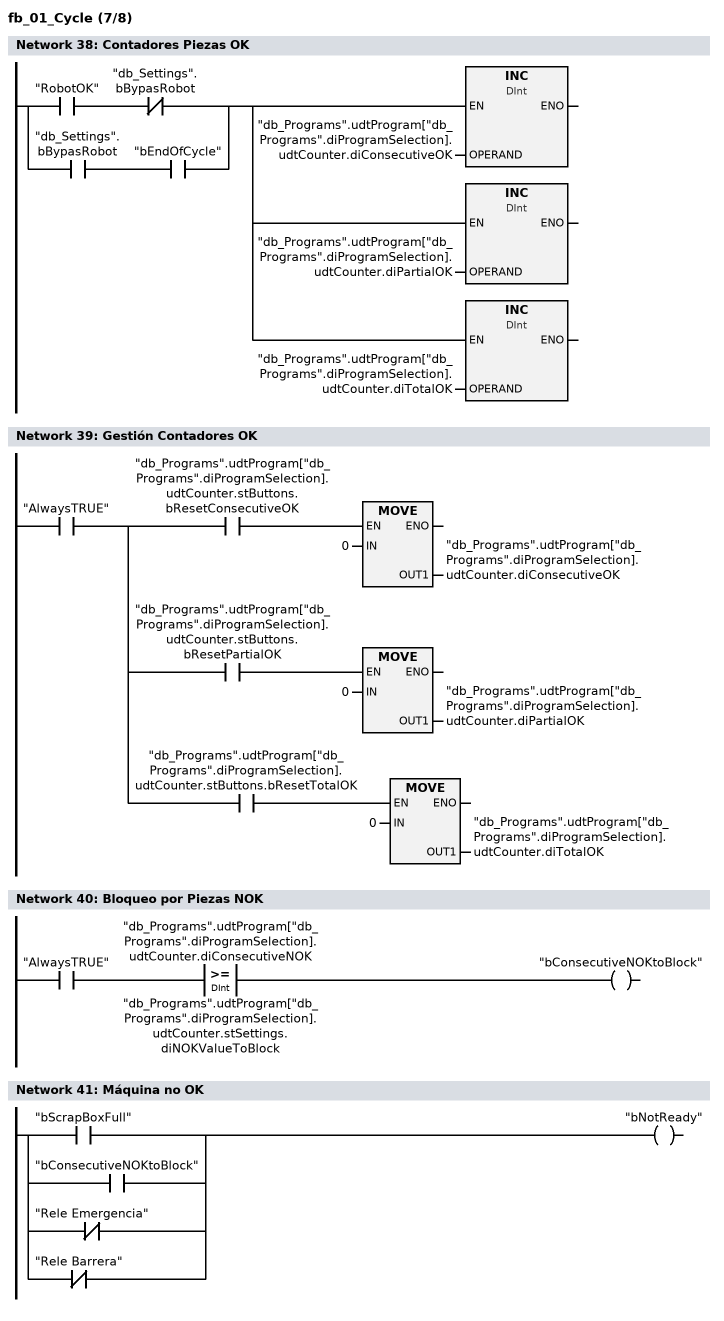
   RUNG wire#powerrail
      Contact( "RobotOK" )
      I_Contact( "db_Settings".bBypasRobot )
      wire#w1
      { S7_Templates := "DestType := DInt" } Inc( "db_Programs".udtProgram["db_Programs".diProgramSelection].udtCounter.diConsecutiveOK )
   END_RUNG
   RUNG wire#powerrail
      Contact( "db_Settings".bBypasRobot )
      Contact( "bEndOfCycle" )
   END_RUNG wire#w1
   RUNG wire#w1
      { S7_Templates := "DestType := DInt" } Inc( "db_Programs".udtProgram["db_Programs".diProgramSelection].udtCounter.diPartialOK )
   END_RUNG
   RUNG wire#w1
      { S7_Templates := "DestType := DInt" } Inc( "db_Programs".udtProgram["db_Programs".diProgramSelection].udtCounter.diTotalOK )
   END_RUNG
   // the same network as SCL:
   IF ("RobotOK" AND NOT "db_Settings".bBypasRobot) OR ("db_Settings".bBypasRobot AND "bEndOfCycle") THEN
       "db_Programs".udtProgram["db_Programs".diProgramSelection].udtCounter.diConsecutiveOK := "db_Programs".udtProgram["db_Programs".diProgramSelection].udtCounter.diConsecutiveOK + 1;
       "db_Programs".udtProgram["db_Programs".diProgramSelection].udtCounter.diPartialOK := "db_Programs".udtProgram["db_Programs".diProgramSelection].udtCounter.diPartialOK + 1;
       "db_Programs".udtProgram["db_Programs".diProgramSelection].udtCounter.diTotalOK := "db_Programs".udtProgram["db_Programs".diProgramSelection].udtCounter.diTotalOK + 1;
   END_IF;
END_REGION

REGION Network 39: Gestión Contadores OK
   RUNG wire#powerrail
      Contact( "AlwaysTRUE" )
      wire#w1
      Contact( "db_Programs".udtProgram["db_Programs".diProgramSelection].udtCounter.stButtons.bResetConsecutiveOK )
      Move(in := 0, out1 => "db_Programs".udtProgram["db_Programs".diProgramSelection].udtCounter.diConsecutiveOK)
   END_RUNG
   RUNG wire#w1
      Contact( "db_Programs".udtProgram["db_Programs".diProgramSelection].udtCounter.stButtons.bResetPartialOK )
      Move(in := 0, out1 => "db_Programs".udtProgram["db_Programs".diProgramSelection].udtCounter.diPartialOK)
   END_RUNG
   RUNG wire#w1
      Contact( "db_Programs".udtProgram["db_Programs".diProgramSelection].udtCounter.stButtons.bResetTotalOK )
      Move(in := 0, out1 => "db_Programs".udtProgram["db_Programs".diProgramSelection].udtCounter.diTotalOK)
   END_RUNG
   // the same network as SCL:
   IF "AlwaysTRUE" AND "db_Programs".udtProgram["db_Programs".diProgramSelection].udtCounter.stButtons.bResetConsecutiveOK THEN
       "db_Programs".udtProgram["db_Programs".diProgramSelection].udtCounter.diConsecutiveOK := 0;
   END_IF;
   IF "AlwaysTRUE" AND "db_Programs".udtProgram["db_Programs".diProgramSelection].udtCounter.stButtons.bResetPartialOK THEN
       "db_Programs".udtProgram["db_Programs".diProgramSelection].udtCounter.diPartialOK := 0;
   END_IF;
   IF "AlwaysTRUE" AND "db_Programs".udtProgram["db_Programs".diProgramSelection].udtCounter.stButtons.bResetTotalOK THEN
       "db_Programs".udtProgram["db_Programs".diProgramSelection].udtCounter.diTotalOK := 0;
   END_IF;
END_REGION

REGION Network 40: Bloqueo por Piezas NOK
   RUNG wire#powerrail
      Contact( "AlwaysTRUE" )
      { S7_Templates := "SrcType := DInt" } GE_Contact(in1 := "db_Programs".udtProgram["db_Programs".diProgramSelection].udtCounter.diConsecutiveNOK, in2 := "db_Programs".udtProgram["db_Programs".diProgramSelection].udtCounter.stSettings.diNOKValueToBlock)
      Coil( "bConsecutiveNOKtoBlock" )
   END_RUNG
   // the same network as SCL:
   "bConsecutiveNOKtoBlock" := "AlwaysTRUE" AND ("db_Programs".udtProgram["db_Programs".diProgramSelection].udtCounter.diConsecutiveNOK >= "db_Programs".udtProgram["db_Programs".diProgramSelection].udtCounter.stSettings.diNOKValueToBlock);
END_REGION

REGION Network 41: Máquina no OK
   RUNG wire#powerrail
      Contact( "bScrapBoxFull" )
      wire#w1
      Coil( "bNotReady" )
   END_RUNG
   RUNG wire#powerrail
      Contact( "bConsecutiveNOKtoBlock" )
   END_RUNG wire#w1
   RUNG wire#powerrail
      I_Contact( "Rele Emergencia" )
   END_RUNG wire#w1
   RUNG wire#powerrail
      I_Contact( "Rele Barrera" )
   END_RUNG wire#w1
   // the same network as SCL:
   "bNotReady" := "bScrapBoxFull" OR "bConsecutiveNOKtoBlock" OR NOT "Rele Emergencia" OR NOT "Rele Barrera";
END_REGION

REGION Network 42: Reset Robot
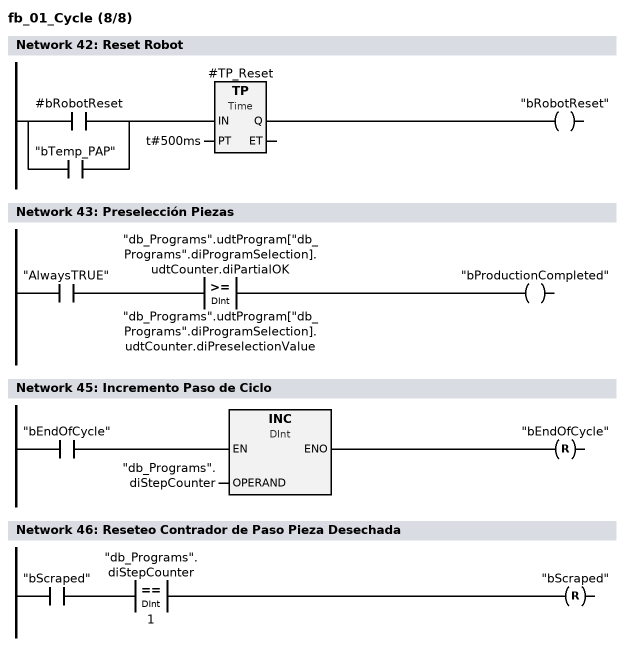
   RUNG wire#powerrail
      Contact( #bRobotReset )
      wire#w1
      { S7_Templates := "time_type := Time" } #TP_Reset.TP(pt := t#500ms, et =>)
      Coil( "bRobotReset" )
   END_RUNG
   RUNG wire#powerrail
      Contact( "bTemp_PAP" )
   END_RUNG wire#w1
   // the same network as SCL:
   #TP_Reset(IN := #bRobotReset OR "bTemp_PAP", PT := t#500ms);   // TP
   "bRobotReset" := #TP_Reset.Q;
END_REGION

REGION Network 43: Preselección Piezas
   RUNG wire#powerrail
      Contact( "AlwaysTRUE" )
      { S7_Templates := "SrcType := DInt" } GE_Contact(in1 := "db_Programs".udtProgram["db_Programs".diProgramSelection].udtCounter.diPartialOK, in2 := "db_Programs".udtProgram["db_Programs".diProgramSelection].udtCounter.diPreselectionValue)
      Coil( "bProductionCompleted" )
   END_RUNG
   // the same network as SCL:
   "bProductionCompleted" := "AlwaysTRUE" AND ("db_Programs".udtProgram["db_Programs".diProgramSelection].udtCounter.diPartialOK >= "db_Programs".udtProgram["db_Programs".diProgramSelection].udtCounter.diPreselectionValue);
END_REGION

REGION Network 45: Incremento Paso de Ciclo
   RUNG wire#powerrail
      Contact( "bEndOfCycle" )
      { S7_Templates := "DestType := DInt" } Inc( "db_Programs".diStepCounter )
      R_Coil( "bEndOfCycle" )
   END_RUNG
   // the same network as SCL:
   IF "bEndOfCycle" THEN
       "db_Programs".diStepCounter := "db_Programs".diStepCounter + 1;
       "bEndOfCycle" := FALSE;
   END_IF;
END_REGION

REGION Network 46: Reseteo Contrador de Paso Pieza Desechada
   RUNG wire#powerrail
      Contact( "bScraped" )
      { S7_Templates := "SrcType := DInt" } EQ_Contact(in1 := "db_Programs".diStepCounter, in2 := 1)
      R_Coil( "bScraped" )
   END_RUNG
   // the same network as SCL:
   IF "bScraped" AND ("db_Programs".diStepCounter = 1) THEN "bScraped" := FALSE; END_IF;
END_REGION
END_FUNCTION_BLOCK
